Staubli VAL3: insert_dOut.pgx

public program insert_dOut(string x_sItem (dimensions=1), bool x_bActive (dimensions=1), dio x_dDio (dimensions=1))
begin
  // insert a new IO
  if isDefined(dOutput[x_sItem])==false and ioStatus(x_dDio)>=0
    insert(dOutput[x_sItem])
    dOutput[x_sItem].bActive=x_bActive
    dOutput[x_sItem].sID=x_sItem
    dOutput[x_sItem].sName=x_sItem
    dioLink(dOutput[x_sItem].dDio,x_dDio)
    dOutput[x_sItem].bEnable=true
  endIf
end
